FUNCTION_BLOCK PnPView_HMI (* Service Interface Function Block Type *)
  (* Standard: 61499-2 *)
  (* Version 0.0, 2/8/2012, XPMUser, nxtControl GmbH, template *)
  PACKAGE Main;
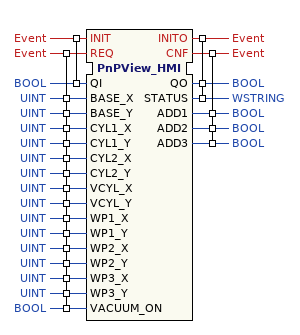
  EVENT_INPUT
    INIT WITH QI;
    REQ WITH BASE_X, BASE_Y, CYL1_X, CYL1_Y, CYL2_X, CYL2_Y, VCYL_X, VCYL_Y, WP1_X, WP1_Y, WP2_X, WP2_Y, WP3_X, WP3_Y, VACUUM_ON;
  END_EVENT
  EVENT_OUTPUT
    INITO WITH QO, STATUS;
    CNF WITH ADD1, ADD2, ADD3;
  END_EVENT
  VAR_INPUT
    QI : BOOL;
    BASE_X : UINT;
    BASE_Y : UINT;
    CYL1_X : UINT;
    CYL1_Y : UINT;
    CYL2_X : UINT;
    CYL2_Y : UINT;
    VCYL_X : UINT;
    VCYL_Y : UINT;
    WP1_X : UINT;
    WP1_Y : UINT;
    WP2_X : UINT;
    WP2_Y : UINT;
    WP3_X : UINT;
    WP3_Y : UINT;
    VACUUM_ON : BOOL;
  END_VAR
  VAR_OUTPUT
    QO : BOOL; (* Event Output Qualifier *)
    STATUS : WSTRING; (* Service Status *)
    ADD1 : BOOL;
    ADD2 : BOOL;
    ADD3 : BOOL;
  END_VAR
END_FUNCTION_BLOCK
